FUNCTION_BLOCK FB_VFormatStr
VAR_INPUT
	sFormat			: STRING(ALARM_TEXT_SIZE);
	pArgStack		: POINTER TO BYTE;
	nStackSize		: DINT;
END_VAR
VAR_OUTPUT
	sOutput			: STRING(ALARM_TEXT_SIZE);
END_VAR
VAR
	fbRdArgStack		: FB_RdArgStack(0, 0);
	nFormatLength		: INT;
	nCurrFormatIndex	: INT;
	nCurrOutputIndex	: INT;
	i					: INT;
	c					: BYTE;
END_VAR
VAR CONSTANT
	SPEC_CHAR	: BYTE := 37;	// '%'
	SPEC_D		: BYTE := 100;	// '%d'
	SPEC_F		: BYTE := 102;	// '%f'
	SPEC_S		: BYTE := 115;	// '%s'
	SPEC_TIME	: BYTE := 84;	// %T
	SPEC_DATE	: BYTE := 68;	// %D
END_VAR

fbRdArgStack.SetMemory(pArgStack, nStackSize);

// Zero output string
F_MemSet(
	pDestAddr:= ADR(sOutput),
	nWithChar:= 0,
	stDestSize:= UDINT_TO_SIZE(SIZEOF(sOutput)));

// Get format string length
nFormatLength := LEN(sFormat);

nCurrFormatIndex := 0;
nCurrOutputIndex := 0;

WHILE NOT AtFmtEnd DO
	
	c := FmtChar;
	NextFmtChar();
	
	IF c = SPEC_CHAR THEN
		
		IF AtFmtEnd THEN
			PutChar(c);
			EXIT;
		END_IF
		
		c := FmtChar;
		NextFmtChar();
	
		CASE c OF
			SPEC_D:
				IF fbRdArgStack.IsIntArg THEN
					PutStr(DINT_TO_STRING(fbRdArgStack.GetIntArg()));
				ELSIF fbRdArgStack.IsUIntArg THEN
					PutStr(UDINT_TO_STRING(fbRdArgStack.GetUIntArg()));
				ELSE
					PutStr('???');
				END_IF
				fbRdArgStack.NextArg();
			SPEC_F:
				IF fbRdArgStack.IsFloatArg THEN
					PutStr(LREAL_TO_STRING(fbRdArgStack.GetFloatArg()));
				ELSE
					PutStr('???');
				END_IF
				fbRdArgStack.NextArg();
			SPEC_S:
				IF fbRdArgStack.IsString THEN
					PutStr(fbRdArgStack.GetStringArg());
				ELSE
					PutStr('???');
				END_IF
			SPEC_TIME:
				IF fbRdArgStack.IsTime THEN
					PutStr(TIME_TO_STRING(fbRdArgStack.GetTimeArg()));
				ELSE
					PutStr('???');
				END_IF
			SPEC_DATE:
				IF fbRdArgStack.IsDate THEN
					PutStr(DATE_TO_STRING(fbRdArgStack.GetDateArg()));
				ELSE
					PutStr('???');
				END_IF			
		ELSE
			IF c = SPEC_CHAR THEN // %% escape sequence?
				PutChar(c);
			ELSE
				PutChar(SPEC_CHAR);
				PutChar(c);
			END_IF
		END_CASE
	ELSE
		PutChar(c);
	END_IF
END_WHILE

PROPERTY PRIVATE AtFmtEnd : BOOL
GET
AtFmtEnd := nCurrFormatIndex >= nFormatLength;
END_GET
END_PROPERTY

PROPERTY PRIVATE FmtChar : BYTE
GET
FmtChar := sFormat[nCurrFormatIndex];
END_GET
END_PROPERTY

METHOD PRIVATE NextFmtChar
VAR_INPUT
END_VAR
IF nCurrFormatIndex < nFormatLength THEN
	nCurrFormatIndex := nCurrFormatIndex + 1;
END_IF
END_METHOD

METHOD PRIVATE PutChar
VAR_INPUT
	nOutChar : BYTE;
END_VAR
IF nCurrOutputIndex < ALARM_TEXT_SIZE THEN
	sOutput[nCurrOutputIndex] := nOutChar;
	nCurrOutputIndex := nCurrOutputIndex + 1;
END_IF
END_METHOD

METHOD PRIVATE PutStr
VAR_INPUT
	sOutStr : STRING(ALARM_TEXT_SIZE);
END_VAR
VAR
	nOutStrLen	: INT;
	i			: INT;
END_VAR
nOutStrLen := LEN(sOutStr);

i := 0;
WHILE i < nOutStrLen AND nCurrOutputIndex < ALARM_TEXT_SIZE DO
	sOutput[nCurrOutputIndex] := sOutStr[i];
	i := i + 1;
	nCurrOutputIndex := nCurrOutputIndex + 1;
END_WHILE
END_METHOD

END_FUNCTION_BLOCK

(* stored: Version 1.1.0.1, ProductVersion 3.1.4024.15
   POU FB_VFormatStr: Id {e1e06578-2e60-4d35-88f4-cf3c69ab23d7}, SpecialFunc None
   Property AtFmtEnd: Id {11da5d1a-43a4-49cc-96cd-82b84905c594}
   Get Get: Id {b5ce0dc0-2eae-443b-a034-59c7c6d102f9}
   Property FmtChar: Id {7c75b97f-dce4-4eb0-91cc-157c47ae4223}
   Get Get: Id {e01712ab-2b4f-417c-a0ec-af6678e4b372}
   Method NextFmtChar: Id {1c40cf68-c45b-49c7-84c2-03d624e16436}
   Method PutChar: Id {eb8931aa-0e28-452e-8931-488be0f8fb85}
   Method PutStr: Id {426bba9e-7651-47bb-9a40-6c30f681f788} *)
